Staubli VAL3: HelloVal3.pjx

--- HelloVal3.pjx ---
Parameters version=s7.9 stackSize=5000 millimeterUnit=true
Program file=start.pgx
Program file=stop.pgx
Data file=HelloVal3.dtx

--- start.pgx ---
program start()
begin
  //1.注释不能写在begin上面
  //2.注释不能写在end下面
  //3.语句后面没有分号也没有冒号

  popUpMsg("Hello world")


end
